FUNCTION BOOLS_TO_ST08X (* this Function combines 8 BOOLS to a 8-BOOL Struct *)
  (* Standard: 61499-1; Description: Copyright (c) 2024 HR Agrartechnik GmbH This program and the accompanying materials are made available under the terms of the Eclipse Public License 2.0 which is available at https://www.eclipse.org/legal/epl-2.0/ SPDX-License-Identifier: EPL-2.0 *)
  (* Version 1.0, 2024-02-22, Franz Höpfinger, HR Agrartechnik GmbH *)
  PACKAGE logiBUS::utils::conversion::str::reversing;
  IMPORT logiBUS::utils::conversion::types::ST08X;
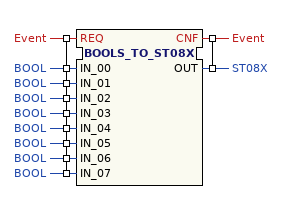
  EVENT_INPUT
    REQ WITH IN_00, IN_01, IN_02, IN_03, IN_04, IN_05, IN_06, IN_07;
  END_EVENT
  EVENT_OUTPUT
    CNF WITH OUT;
  END_EVENT
  VAR_INPUT
    IN_00 : BOOL; (* BIT 00 *)
    IN_01 : BOOL; (* BIT 01 *)
    IN_02 : BOOL; (* BIT 02 *)
    IN_03 : BOOL; (* BIT 03 *)
    IN_04 : BOOL; (* BIT 04 *)
    IN_05 : BOOL; (* BIT 05 *)
    IN_06 : BOOL; (* BIT 06 *)
    IN_07 : BOOL; (* BIT 07 *)
  END_VAR
  VAR_OUTPUT
    OUT : logiBUS::utils::conversion::types::ST08X; (* ST08X Output *)
  END_VAR
  BODY IN ST:
PACKAGE logiBUS::utils::conversion::str::reversing;

IMPORT logiBUS::utils::conversion::types::ST08X;

(* this Function combines 8 BOOLS to a 8-BOOL Struct *)
FUNCTION BOOLS_TO_ST08X

VAR_INPUT
	IN_00 : BOOL; // BIT 00
	IN_01 : BOOL; // BIT 01
	IN_02 : BOOL; // BIT 02
	IN_03 : BOOL; // BIT 03
	IN_04 : BOOL; // BIT 04
	IN_05 : BOOL; // BIT 05
	IN_06 : BOOL; // BIT 06
	IN_07 : BOOL; // BIT 07
END_VAR

VAR_OUTPUT
	OUT : ST08X; // ST08X Output
END_VAR

OUT.X_00 := IN_00;
OUT.X_01 := IN_01;
OUT.X_02 := IN_02;
OUT.X_03 := IN_03;
OUT.X_04 := IN_04;
OUT.X_05 := IN_05;
OUT.X_06 := IN_06;
OUT.X_07 := IN_07;

END_FUNCTION
  END_BODY
END_FUNCTION
